// TIA Portal V19 export
TYPE "udt_DoorSts"
// stored: Access Published, IsFailsafeCompliant true
   STRUCT
      OK : Bool;   // Door closed and restored
      NormalStop : Bool;   // Entry request
      SafeStop : Bool;   // Door Open
      EntryEnable : Bool;   // Door Entry Enable
      Warning_DoorOpened : Bool;   // Door opening in progress
      Warning_DoorOpenRequest : Bool;   // Door opening in progress
   END_STRUCT;
END_TYPE
